# EPICS substitutions: db/Beckhoff_7XXX/ecmcEL7041-1000.substitutions
file "ecmcEcSlave.template"
{
  pattern {}
          {}
}

file "ecmcEL7037-chX.template"
{
  pattern {CH_ID}
          {01   }
}

file "ecmcEL5101-chX.template"
{
  pattern {CH_ID}
          {01   }
}
